// Implicitly generated code : DO NOT EDIT
FUNCTION CheckLRangeUnsigned : ULINT
VAR_INPUT
	value, lower, upper: ULINT;
END_VAR

// Implicitly generated code : Only an Implementation suggestion
{noflow}
Fault_Count_G(CU:=FALSE) ; 
IF (value < lower) THEN
	CheckLRangeUnsigned := lower;
		Fault_Count_G(CU:=TRUE) ; 
ELSIF(value > upper) THEN
	CheckLRangeUnsigned := upper;
		Fault_Count_G(CU:=TRUE) ; 
ELSE
	CheckLRangeUnsigned := value;
END_IF
{flow}

END_FUNCTION

(* stored: Version 1.1.0.1, ProductVersion 3.1.4024.2
   POU CheckLRangeUnsigned: Id {890a5ad9-473f-4314-99f4-768799f44efe}, SpecialFunc CheckLRangeUnsigned *)
